Staubli VAL3: saveTrack.dtx

public aio aEncoder = {link=e01CurrPos}
public aio aEncoderLatch = {link=ModbusSrv-0\Modbus-Word\encoder}
public aio aEncoderSpeed = {link=ModbusSrv-0\Modbus-Word\encoder}
public aio e00Counts = {link=e00Counts}
public aio e00CountsMes = {link=e00CountsMes}
public aio e00CurrPos = {link=e01CurrPos}
public aio e00LatchFilter = {link=e00LatchFilter}
public aio e00LatchPos = {link=e01LatchPos}
public aio e00PrstPos = {link=e00PrstPos}
public aio e01CurrPos = {link=e01CurrPos}
public aio e01LatchPos = {link=e01LatchPos}
public aio enc_speed = {link=ModbusSrv-0\Modbus-Word\speed}
public bool bAlreadyStart
public bool bRemoveOnStop = true
public bool bResetOnStart = true
public bool bSimulate
public bool bTrackLoad
public bool bUseFrontUP = true
dio MbIn[8] = {link=ModbusSrv-0\Modbus-Bit\MbIn[0]}
public dio dEnableLatch = {link=e01EnLatch}
public dio dLatchInput = {link=e01LatchSig}
public dio e00CountsErr = {link=e00CountsErr}
public dio e00EnLatch = {link=e01EnLatch}
public dio e00EnPrst = {link=e00EnPrst}
public dio e00HwErr = {link=e00HwErr}
public dio e00Latch = {link=e00Latch}
public dio e00LatchEdgFall = {link=e00LatchEdgFall}
public dio e00LatchSig = {link=e01LatchSig}
public dio e00OvsErr = {link=e00OvsErr}
public dio e00PowerErr = {link=e00PowerErr}
public dio e00RstErr = {link=e00RstErr}
public dio e01EnLatch = {link=e01EnLatch}
public dio e01Latch = {link=e01Latch}
public dio e01LatchSig = {link=e01LatchSig}
public dio valve1 = {link=valve1}
public mdesc mNomSpeed = {blend=off}
public num nAcc = 200
public num nENCSCALEFACTOR
public num nFilterSize = 50
public num nFilterTime = 4
public num nIndexGun = 1
public num nMAXCOUNT = 65535
public num nOffsetDistance
public num nOffsetLimit = 500
public num nSensor2Win
public num nSensorDelay = 1
public num nSensorDist = 100
public num nSensorPeriod = 1
public num nSimulateSpeed = 30
public num nStabTime
public num nStackSize = 6
public num nTimeOff = -1
public num nTrackSmooth = 5
public pointRx pWinConvPlane = {x=768.558802, y=425.100094, z=-259.30763, rx=0.006936, ry=-179.488005, rz=0.33162, shoulder=lefty, elbow=epositive, wrist=wpositive, fatherId=world[0]}
public pointRx pWinDownLim = {x=713.971282, y=425.100121, z=-259.307641, rx=0.007248, ry=-179.487322, rz=0.331196, shoulder=lefty, elbow=epositive, wrist=wpositive, fatherId=world[0]}
public pointRx pWinUpLim = {x=711.850001, y=-407.745087, z=-259.307675, rx=0.00642, ry=-179.486136, rz=0.33201, shoulder=lefty, elbow=epositive, wrist=wpositive, fatherId=world[0]}
public tool tGun = {fatherId=flange[0], ioLink=valve1}
public aio e01Counts = {link=e01Counts}
public dio e01CountsErr = {link=e01CountsErr}
public aio e01CountsMes = {link=e01CountsMes}
public dio e01EnPrst = {link=e01EnPrst}
public dio e01HwErr = {link=e01HwErr}
public dio e01LatchEdgFall = {link=e01LatchEdgFall}
public aio e01LatchFilter = {link=e01LatchFilter}
public dio e01OvsErr = {link=e01OvsErr}
public dio e01PowerErr = {link=e01PowerErr}
public aio e01PrstPos = {link=e01PrstPos}
public dio e01RstErr = {link=e01RstErr}
